{attribute 'GeneratedUsingTerminal: EK1121-0010-0016'}
{attribute addProperty BoxType "EK1121-0010-0016"}
{attribute addProperty Id "InfoDataAT %I*InfoData_6F19DB2B2"}
{attribute addProperty CRC "532711307"}
{attribute addProperty Size "2"}
TYPE EK1121_1FC0878B EXTENDS EtcSlaveTerminalBase_947E5A46 :
STRUCT
	{attribute addProperty Name "InfoData"}
	InfoData : InfoData_6F19DB2B;
END_STRUCT
END_TYPE

(* stored: Version 1.2.0.0, ProductVersion 3.1.4024.9
   DUT EK1121_1FC0878B: Id {d4e2e7be-f590-43bc-96d1-fbab6e22d9da} *)
